INTERFACE I_Deserializable

METHOD TryDeserializeWith : BOOL
VAR_INPUT
	Deserializer : I_Deserializer;
END_VAR
END_METHOD

END_INTERFACE

(* stored: Version 1.1.0.1, ProductVersion 3.1.4024.12
   Itf I_Deserializable: Id {86c365a9-0310-4af1-8eef-306315ca97b2}
   Method TryDeserializeWith: Id {dafd7abe-c1cd-45fb-97d9-cf4c65d26eb4} *)
